(* IEC 61131-3 sources: LASAL/Class/CommandServer, 1 file *)

(* ---- CommandServer.st ---- *)
(*!
<Class
	Name               = "CommandServer"
	Revision           = "0.0"
	RealtimeTask       = "false"
	CyclicTask         = "true"
	DefCyclictime      = "10 ms"
	BackgroundTask     = "false"
	Sigmatek           = "false"
	OSInterface        = "false"
	HighPriority       = "false"
	Automatic          = "false"
	UpdateMode         = "Prescan"
	SharedCommandTable = "true"
	Objectsize         = "(750,360)">
	<Channels>
		<Client Name="CmdRouter" Required="true" Internal="false"/>
	</Channels>
	<Network Name="CommandServer">
		<!-- List of Components in this network -->
		<Components>
			<Object
				Name       = "_base"
				Class      = "_TCPIP_SERVER"
				Position   = "(218,120)"
				Visualized = "true"
				Remotely   = "true">
				<Channels>
					<Server Name="sControl"/>
					<Server Name="SemaName01"/>
					<Server Name="SemaName02"/>
					<Server Name="sError"/>
					<Server Name="TaskName"/>
					<Client Name="cConfig"/>
					<Client Name="cMaxConnections" Value="0"/>
					<Client Name="co_MultiTask"/>
					<Client Name="co_SigCLib"/>
					<Client Name="co_StdLib"/>
					<Client Name="co_Task"/>
					<Client Name="cPort"/>
					<Client Name="cSizeOfTXBuffer"/>
					<Client Name="cTimeout"/>
				</Channels>
			</Object>
		</Components>
		<Comments>
		</Comments>
		<!-- List of Connections in this network -->
		<Connections>
			<Connection Source="this.sControl" Destination="_base.sControl" Vertices="(996,210),(824,210),"/>
			<Connection Source="this.sError" Destination="_base.sError" Vertices="(996,270),(824,270),"/>
			<Connection Source="this.TaskName" Destination="_base.TaskName" Vertices="(996,330),(824,330),"/>
			<Connection Source="this.SemaName01" Destination="_base.SemaName01" Vertices="(996,390),(824,390),"/>
			<Connection Source="this.SemaName02" Destination="_base.SemaName02" Vertices="(996,450),(824,450),"/>
		</Connections>
		<!-- Headerfiles -->
		<Options>
		</Options>
	</Network>
</Class>
*)
#pragma using _TCPIP_SERVER

CommandServer : CLASS
: _TCPIP_SERVER
  //Servers:
  //Clients:
	CmdRouter 	: CltChCmd_CommandRouter;
  //Variables:
		sendBuffer : ARRAY [0..1024] OF CHAR;

		Socket 	: DINT;
  //Functions:
				//! <Function Comment="This Method is called if Data is received (Overwrite it, to create a Request)" Name="Response"/>
	FUNCTION VIRTUAL GLOBAL Response
		VAR_INPUT
			pData 	: ^void;			//! <Variable Comment="Pointer to Data" Name="Response.pData"/>
			udSize 	: UDINT;			//! <Variable Comment="Size of Data" Name="Response.udSize"/>
			dSock 	: DINT;			//! <Variable Comment="Socketnumber" Name="Response.dSock"/>
		END_VAR;

	FUNCTION GLOBAL SendStatus
		VAR_INPUT
			Status 	: DINT;
		END_VAR;
  //Tables:
	FUNCTION @STD
		VAR_OUTPUT
			ret_code	: CONFSTATES;
		END_VAR;
	FUNCTION GLOBAL TAB @CT_;
END_CLASS;

#pragma usingLtd CommandRouter

(* CommandServer::Response
Inherited method: The method is over-written to allow for the incoming
data to be read.
*)
FUNCTION VIRTUAL GLOBAL CommandServer::Response
	VAR_INPUT
    // pointer to the data buffer
		pData 	: ^void;
    // size of the data received
		udSize 	: UDINT;
    // socket number from which data was received
		dSock 	: DINT;
	END_VAR
  VAR
  	pSendData : CHAR;
  END_VAR

  Socket:=dSock;

  CmdRouter.SetData(pData:=pData,size:=udSize);

//  sendBuffer[0] := 'A';
//  sendBuffer[1] := 'C';
//  sendBuffer[2] := 'K';
//
//  SendData(pData:=#sendBuffer[0], udSize:=3, dSock:=dSock, bDirect:=0);

END_FUNCTION

FUNCTION GLOBAL CommandServer::SendStatus
	VAR_INPUT
		Status 	: DINT;
	END_VAR

  sendBuffer[0] := 'A';
  sendBuffer[1] := 'C';
  sendBuffer[2] := 'K';

  SendData(pData:=#sendBuffer[0], udSize:=3, dSock:=Socket, bDirect:=1);

END_FUNCTION
